// TIA Portal project "Test_SCL" (V15.1)

(* hardware
DEVICE "S71500/ET200MP station_1"  S7-1500 station
   slot 0: "Rail_0"  Rack  6ES7 590-1***0-0AA0
   slot 1: "PLC_1"  CPU 1513-1 PN  6ES7 513-1AL02-0AB0  V2.6
      slot 3: "CPU display_1"  6ES7591-1AA00-0AA0
*)

// ===== PLC "PLC_1"  CPU 1513-1 PN =====

VAR_GLOBAL   // PLC tag table "Default tag table"
   "Clock_Byte" AT %MB0 : Byte;
   "Clock_10Hz" AT %M0.0 : Bool;
   "Clock_5Hz" AT %M0.1 : Bool;
   "Clock_2.5Hz" AT %M0.2 : Bool;
   "Clock_2Hz" AT %M0.3 : Bool;
   "Clock_1.25Hz" AT %M0.4 : Bool;
   "Clock_1Hz" AT %M0.5 : Bool;
   "Clock_0.625Hz" AT %M0.6 : Bool;
   "Clock_0.5Hz" AT %M0.7 : Bool;
END_VAR

DATA_BLOCK "Data"   // DB1
{ S7_Optimized_Access := 'TRUE' }
VERSION : 0.1
   VAR
      nr_1 : Int;
      nr_2 : Int;
      nr_3 : Int;
      nr_4 : Int;
      nr_re_1 : Real;
      nr_re_2 : Real;
      nr_re_3 : Real;
      nr_re_4 : Real;
      put_in : Bool;
      take_out : Bool;
      select_shelf : Int;
      error : Bool;
      counter_for : Int;
      shelf : Array[0..99] of Bool;
      erase : Bool;
      cond_while : Bool := true;
      counter_while : Int;
      led_state : Int;
      led_color : String;
      nr_a : Int;
      nr_b : Int;
      cmmdc : Int;
      cmmmc : Int;
      aux_cmmmc_1 : Int;
      aux_cmmmc_2 : Int;
   END_VAR
BEGIN
END_DATA_BLOCK

DATA_BLOCK "Binary_Search"   // DB2
{ S7_Optimized_Access := 'TRUE' }
VERSION : 0.1
   VAR
      array_sortat : Array[0..9] of Int;
      left : Int;
      right : Int := 9;
      middle : Int;
      value_search : Int := 6;
      start : Bool;
   END_VAR
BEGIN
   array_sortat[0] := 1;
   array_sortat[1] := 2;
   array_sortat[2] := 3;
   array_sortat[3] := 4;
   array_sortat[4] := 5;
   array_sortat[5] := 6;
   array_sortat[6] := 7;
   array_sortat[7] := 8;
   array_sortat[8] := 9;
   array_sortat[9] := 10;
END_DATA_BLOCK

DATA_BLOCK "Sortare"   // DB3
{ S7_Optimized_Access := 'TRUE' }
VERSION : 0.1
   VAR
      "array" : Array[0..9] of Int;
      index : Int;
      aux : Int;
      counter_for_1 : Int;
      counter_for_2 : Int;
      swap : Bool;
      start : Bool;
   END_VAR
BEGIN
   "array"[0] := 5;
   "array"[1] := 6;
   "array"[3] := 7;
   "array"[2] := 3;
   "array"[5] := 4;
   "array"[4] := 1;
   "array"[6] := 2;
   "array"[7] := 9;
   "array"[8] := 8;
   "array"[9] := 10;
END_DATA_BLOCK

ORGANIZATION_BLOCK "Main"   // OB1, LAD, ProgramCycle
TITLE = "Main Program Sweep (Cycle)"
{ S7_Optimized_Access := 'TRUE' }
VERSION : 0.1
   VAR_INPUT
      Initial_Call : Bool;   // Initial call of this OB
      Remanence : Bool;   // =True, if remanent data are available
   END_VAR
BEGIN

REGION Network 1 (SCL): Simple math examples
   "Data".nr_1 := 20;
   "Data".nr_2 := 16;
   "Data".nr_re_2 := 16.4;
   "Data".nr_4 := 2;
   "Data".nr_3 := "Data".nr_1 MOD "Data".nr_2;
   "Data".nr_re_1 := "Data".nr_re_2 * "Data".nr_re_2;
   "Data".nr_re_3 := INT_TO_REAL("Data".nr_1) ** "Data".nr_4;

   "Data".nr_1 += 1;
END_REGION

REGION Network 2 (SCL): if, then, else, elsif
   IF "Data".put_in AND "Data".take_out = FALSE THEN
       // Statement section IF
       "Data".shelf["Data".select_shelf] := TRUE;
   ELSIF "Data".take_out AND "Data".put_in = FALSE THEN
       "Data".shelf["Data".select_shelf] := FALSE;
   ELSIF "Data".take_out AND "Data".put_in THEN
       "Data".error := TRUE;
   ELSE
       "Data".error := FALSE;
   END_IF;
END_REGION

REGION Network 3 (SCL): for, while
   IF "Data".erase = TRUE THEN
       // Statement section IF
       FOR "Data".counter_for := 0 TO 99 DO
           // Statement section FOR
           "Data".shelf["Data".counter_for] := FALSE;
       END_FOR;
   END_IF;

   //to do an "even" for loop
   //FOR "Data".counter_for := 0 TO 99 BY 2 DO

   WHILE "Data".cond_while DO
       // Statement section WHILE
       IF "Data".counter_while MOD 2 = 0 THEN
           "Data".shelf["Data".counter_while] := TRUE;
       ELSE
           "Data".shelf["Data".counter_while] := FALSE;
       END_IF;
       "Data".counter_while += 1;
       IF "Data".counter_while > 99 THEN
           "Data".cond_while := FALSE;
       END_IF;
   END_WHILE;

   (*
   WHILE "Data".counter_while <= 99 DO
       // Statement section WHILE
       IF "Data".counter_while MOD 2 = 0 THEN
           "Data".shelf["Data".counter_while] := TRUE;
       ELSE
           "Data".shelf["Data".counter_while] := FALSE;
       END_IF;
       "Data".counter_while += 1;
   END_WHILE;
   *)

   "Data".counter_while := 0;
END_REGION

REGION Network 4 (SCL): case
   CASE "Data".led_state OF
       1:
           "Data".led_color := 'Red';
           //RETURN
       2:
           "Data".led_color := 'Green';
           //RETURN
       3:
           "Data".led_color := 'Blue';
           //RETURN
       ELSE  // Statement section ELSE
           "Data".led_color := 'Off';
   END_CASE;

   //RETURN doar iese de tot din switch case
END_REGION

REGION Network 5 (SCL): cmmdc
   (*
   IF "Data".nr_a > "Data".nr_b THEN
       "Data".aux_cmmdc := "Data".nr_a;
       "Data".nr_b := "Data".nr_a;
       "Data".nr_a := "Data".aux_cmmdc;
   END_IF;
   *)

   "Data".nr_a := 20;
   "Data".nr_b := 16;

   WHILE "Data".nr_a <> "Data".nr_b DO
       IF "Data".nr_a > "Data".nr_b THEN
           "Data".nr_a -= "Data".nr_b;
       ELSE
           "Data".nr_b -= "Data".nr_a;
       END_IF;
   END_WHILE;
END_REGION

REGION Network 6 (SCL): cmmmc
   "Data".nr_a := 10;
   "Data".nr_b := 18;

   "Data".aux_cmmmc_1 := "Data".nr_a;
   "Data".aux_cmmmc_2 := "Data".nr_b;

   WHILE "Data".aux_cmmmc_1 <> "Data".aux_cmmmc_2 DO
       IF "Data".aux_cmmmc_1 < "Data".aux_cmmmc_2 THEN
           "Data".aux_cmmmc_1 += "Data".nr_a;
       ELSE
           "Data".aux_cmmmc_2 += "Data".nr_b;
       END_IF;
   END_WHILE;
END_REGION

REGION Network 7 (SCL): Binary search
   IF "Binary_Search".start = True THEN
       WHILE "Binary_Search".array_sortat["Binary_Search".middle] <> "Binary_Search".value_search DO
           "Binary_Search".middle := ("Binary_Search".left + "Binary_Search".right) / 2;
           IF "Binary_Search".array_sortat["Binary_Search".middle] < "Binary_Search".value_search THEN
               "Binary_Search".left := "Binary_Search".middle + 1;
           ELSIF "Binary_Search".array_sortat["Binary_Search".middle] > "Binary_Search".value_search THEN
               "Binary_Search".right := "Binary_Search".middle - 1;
           ELSE
               "Binary_Search".start := false;
               RETURN;
           END_IF;
       END_WHILE;
   ELSE
       "Binary_Search".left := 0;
       "Binary_Search".right := 9;
   END_IF;
END_REGION

REGION Network 8 (SCL): Sortare
   IF "Sortare".start = TRUE THEN
       FOR "Sortare".counter_for_1 := 0 TO 9 DO
           "Sortare".swap := FALSE;
           FOR "Sortare".counter_for_2 := 0 TO 8 - "Sortare".counter_for_1 DO
               IF "Sortare".array["Sortare".counter_for_2] > "Sortare".array["Sortare".counter_for_2 + 1] THEN
                   "Sortare".aux := "Sortare".array["Sortare".counter_for_2];
                   "Sortare".array["Sortare".counter_for_2] := "Sortare".array["Sortare".counter_for_2 + 1];
                   "Sortare".array["Sortare".counter_for_2 + 1] := "Sortare".aux;
                   "Sortare".swap := TRUE;
               END_IF;
           END_FOR;
           IF "Sortare".swap = FALSE THEN
               "Sortare".start := FALSE;
               EXIT;
           END_IF;
       END_FOR;
       "Sortare".start := FALSE;
   END_IF;
END_REGION
END_ORGANIZATION_BLOCK